// TIA Portal V20 export
TYPE "LKinCtrl_typePathData_reduced"
   STRUCT
      pathDataName : String["LKINCTRL_LENGTH_OF_PATHDATA_NAME"];   // name of PathData
      commands : Array[1.."LKINCTRL_NO_OF_PATHDATA_ELEMENTS_REDUCED"] of "LKinCtrl_typePathDataElement_reduced";   // command list
   END_STRUCT;
   // commands[1].cmdParameters.transitionParameters[1] := -1.0;
   // commands[2].cmdParameters.transitionParameters[1] := -1.0;
   // commands[3].cmdParameters.transitionParameters[1] := -1.0;
   // commands[4].cmdParameters.transitionParameters[1] := -1.0;
   // commands[5].cmdParameters.transitionParameters[1] := -1.0;
   // commands[6].cmdParameters.transitionParameters[1] := -1.0;
   // commands[7].cmdParameters.transitionParameters[1] := -1.0;
   // commands[8].cmdParameters.transitionParameters[1] := -1.0;
   // commands[9].cmdParameters.transitionParameters[1] := -1.0;
   // commands[10].cmdParameters.transitionParameters[1] := -1.0;
END_TYPE
